// Mitsubishi GX Works2 project: encoEx01   PLC: Q02/Q02H

PROGRAM MAIN
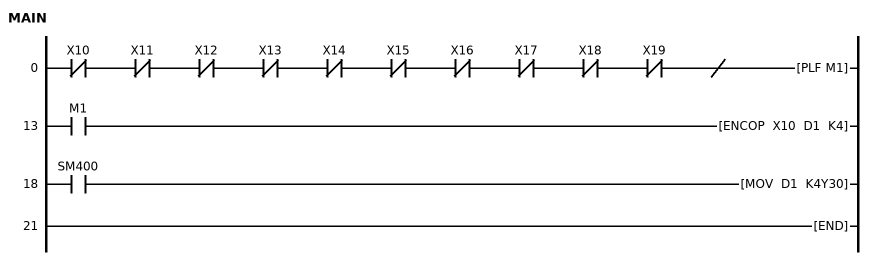
0     LDI     X10
      ANI     X11
      ANI     X12
      ANI     X13
      ANI     X14
      ANI     X15
      ANI     X16
      ANI     X17
      ANI     X18
      ANI     X19
      INV
      PLF     M1
13    LD      M1
      ENCOP   X10 D1 K4
18    LD      SM400
      MOV     D1 K4Y30
21    END
END_PROGRAM
